TYPE ST_General :
STRUCT
	AcknowledgeAllCmd : BOOL;
	
END_STRUCT
END_TYPE

(* stored: Version 1.1.0.1, ProductVersion 3.1.4024.5
   DUT ST_General: Id {a39d0f48-12cf-4fdb-ab91-05df24c1c258} *)
